(* IEC 61131-3 sources: traffic-lights/PLC_TrafficLights/Class/Random, 1 file *)

(* ---- Random.st ---- *)
#DEFINE MULTIPLIER  11035152
#DEFINE INCREMENT 12345
#DEFINE MODULUS 214748364

(*!
<Class
	Name               = "Random"
	Revision           = "0.0"
	RealtimeTask       = "false"
	CyclicTask         = "false"
	BackgroundTask     = "false"
	Sigmatek           = "false"
	OSInterface        = "false"
	HighPriority       = "false"
	Automatic          = "false"
	UpdateMode         = "Prescan"
	SharedCommandTable = "true"
	Objectsize         = "(284,120)">
	<Channels>
		<Server Name="ClassSvr" Visualized="false" Initialize="false" WriteProtected="true" Retentive="false"/>
	</Channels>
</Class>
*)
Random : CLASS
  //Servers:
	ClassSvr 	: SvrChCmd_DINT;
  //Clients:
  //Variables:
		Seed 	: UDINT;
  //Functions:

	FUNCTION GLOBAL GetRandomNumber
		VAR_INPUT
			Minimum 	: DINT;
			Maximum 	: DINT;
		END_VAR
		VAR_OUTPUT
			RandomNumber 	: DINT;
		END_VAR;
  //Tables:
	FUNCTION @STD
		VAR_OUTPUT
			ret_code	: CONFSTATES;
		END_VAR;
	FUNCTION GLOBAL TAB @CT_;
END_CLASS;

//----------------------------------------------------------------------------------------------------
//  Externally called methods
//----------------------------------------------------------------------------------------------------

FUNCTION GLOBAL Random::GetRandomNumber
	VAR_INPUT
		Minimum 	: DINT;
		Maximum 	: DINT;
	END_VAR
	VAR_OUTPUT
		RandomNumber 	: DINT;
	END_VAR

    IF Seed = 0 THEN
        Seed := 123;
    END_IF;

    // This algorithm is a Linear congruential generator (LCG).
    // Not safe for uses relating to security.
    Seed := (MULTIPLIER * Seed + INCREMENT) MOD MODULUS;
    RandomNumber := Minimum + (TO_DINT(Seed) MOD (Maximum - Minimum + 1));

END_FUNCTION
